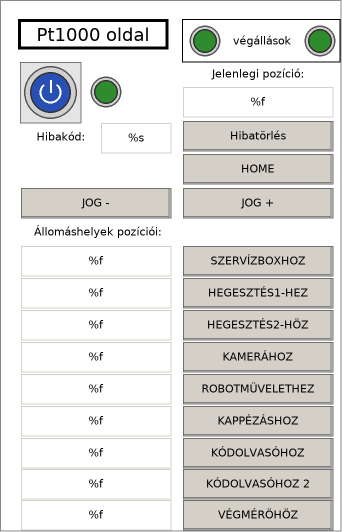
VISUALIZATION Tengely_Pt1000  // 342x532
    PowerSwitch (20,62 61x61), variable: GVL.bPistiServo, behaviour: TOGGLE, style: Switch-PowerSwitch-Blue
    Button (183,154 150x30), "HOME"
        OnMouseUp: execute { PISTITENGELY.sPistiAxisCommand:='HOME'; }
    Button (183,188 150x30), "JOG +"
        tap PISTITENGELY.bPistiJOGPlus
    Button (21,188 150x30), "JOG -"
        tap PISTITENGELY.bPistiJOGMinus
    Button (183,121 150x30), "Hibatörlés"
        tap PISTITENGELY.bPistiReset
    Textfield (101,123 70x30), "%s", text variable: PISTITENGELY.nPistiErrorCode, input disabled if: TRUE
    Textfield (21,310 150x30), "%f", text variable: GVL.lrHegesztoPosition7
    Button (183,310 150x30), "HEGESZTÉS2-HÖZ"
        OnMouseUp: execute { PISTITENGELY.lrPistiPosition:=GVL.lrHegesztoPosition7; PISTITENGELY.sPistiAxisCommand:='MOVE'; }
    Label (183,64 150x20), "Jelenlegi pozíció:"
    Textfield (183,87 150x30), "%f", text variable: PISTITENGELY.lrPistiActPos, input disabled if: TRUE
    Button (183,246 150x30), "SZERVÍZBOXHOZ"
        OnMouseUp: execute { PISTITENGELY.lrPistiPosition:=GVL.lrPtSzervizbox; PISTITENGELY.sPistiAxisCommand:='MOVE'; }
    Textfield (21,246 150x30), "%f", text variable: GVL.lrPtSzervizbox
    Textfield (21,278 150x30), "%f", text variable: GVL.lrHegesztoPosition6
    Button (183,278 150x30), "HEGESZTÉS1-HEZ"
        OnMouseUp: execute { PISTITENGELY.lrPistiPosition:=GVL.lrHegesztoPosition6; PISTITENGELY.sPistiAxisCommand:='MOVE'; }
    Lamp1 (88,74 36x36), variable: PISTITENGELY.bHomeReady, style: Lamp-Lamp1-Green
    RoundedRectangle (18,19 150x30)
    Label (18,20 150x30), "Pt1000 oldal"
    Textfield (21,374 150x30), "%f", text variable: GVL.lrRobotKappePosition
    Button (183,374 150x30), "ROBOTMÜVELETHEZ"
        OnMouseUp: execute { PISTITENGELY.lrPistiPosition:=GVL.lrRobotKappePosition; PISTITENGELY.sPistiAxisCommand:='MOVE'; }
    Textfield (21,500 150x30), "%f", text variable: GVL.lrVegmeroPosition
    Button (183,500 150x30), "VÉGMÉRÖHÖZ"
        OnMouseUp: execute { PISTITENGELY.lrPistiPosition:=GVL.lrVegmeroPosition; PISTITENGELY.sPistiAxisCommand:='MOVE'; }
    Textfield (21,406 150x30), "%f", text variable: GVL.lrKappePosition
    Button (183,406 150x30), "KAPPÉZÁSHOZ"
        OnMouseUp: execute { PISTITENGELY.lrPistiPosition:=GVL.lrKappePosition; PISTITENGELY.sPistiAxisCommand:='MOVE'; }
    Textfield (21,438 150x30), "%f", text variable: GVL.lrKodolvasasPosition
    Button (183,438 150x30), "KÓDOLVASÓHOZ"
        OnMouseUp: execute { PISTITENGELY.lrPistiPosition:=GVL.lrKodolvasasPosition; PISTITENGELY.sPistiAxisCommand:='MOVE'; }
    Label (26,127 70x20), "Hibakód:"
    Label (23,222 150x20), "Állomáshelyek pozíciói:"
    Group (182,19 158x43)
        Rectangle (0,0 158x43)
        Lamp1 (5,4 36x36), variable: GVL.bPistiNegSwitch, style: Lamp-Lamp1-Green
        Lamp1 (120,4 36x36), variable: GVL.bPistiPosSwitch, style: Lamp-Lamp1-Green
        Label (45,12 70x20), "végállások"
    Textfield (21,342 150x30), "%f", text variable: GVL.lrPtKameraPosition
    Button (183,342 150x30), "KAMERÁHOZ"
        OnMouseUp: execute { PISTITENGELY.lrPistiPosition:=GVL.lrPtKameraPosition; PISTITENGELY.sPistiAxisCommand:='MOVE'; }
    Textfield (21,469 150x30), "%f", text variable: GVL.lrKodolvasasPosition2
    Button (183,469 150x30), "KÓDOLVASÓHOZ 2"
        OnMouseUp: execute { PISTITENGELY.lrPistiPosition:=GVL.lrKodolvasasPosition2; PISTITENGELY.sPistiAxisCommand:='MOVE'; }
END_VISUALIZATION

(* stored: Version 1.1.0.1, ProductVersion 3.1.4024.11
   Visu Tengely_Pt1000: Id {f52d2f44-c0ec-4c3f-825c-817e810dc813} *)
